PROGRAM S09_CardCarrying
VAR
	//工站
	station					: REFERENCE TO FB_Station:=fbstation[9];
	//气缸
	fbHOZCyl	:REFERENCE TO FB_Cylinder:=fbCylinder[33];	//	卡片上料Y轴气缸
	fbVTCCyl_1	:REFERENCE TO FB_Cylinder:=fbCylinder[34];	//	卡片上料Z轴气缸1(上)
	fbVTCCyl_2	:REFERENCE TO FB_Cylinder:=fbCylinder[35];	//	卡片上料Z轴气缸2（下）



	//伺服
	fbROTAxisMove	 :REFERENCE TO FB_Axis:=fbAxis[16];	//	出料线体伺服
	fbZAxisStepMotor1	 :REFERENCE TO FB_Axis:=fbAxis[17];	//	卡片顶升步进
	fbZAxisStepMotor2	 :REFERENCE TO FB_Axis:=fbAxis[18];	//	卡片顶升步进
	


	
	//延时
	arTonDelay :ARRAY[1..20] OF TON;
	//返回值
	UdiReturnValue :ARRAY[1..20] OF UDINT;
	//过程记录
	tsModuleProcess:ARRAY[1..gc_ModuleProNo] OF DUT_Process;
	xClearModuleProcessDone:BOOL;
	bClearProcessStep	:BYTE;
	i: INT;
	
	// //破真空
	xVacuum_BreakValveControl:ARRAY[1..2]OF BOOL;
	// //破真空完成
	xVacuum_BreakCompleted:ARRAY[1..2] OF BOOL;
	// //卡片到位传感器
	xCardSensorReached: ARRAY[1..2] of bool;
	// //卡片存在检测
	xCardCheckSensor: ARRAY[1..2] of bool;
	
	 //报警屏蔽
	_AlarmDisable: BOOL;
	// //真空吸动作
	xVacuum_WorkValveControl: ARRAY[1..2] OF BOOL;
	// //真空吸到达真空
	xVacuumWorkCompleted:ARRAY[1..2] OF BOOL;
	// //皮带线上检测卡片
	xBeltCardCheckSensor:ARRAY[1..2] OF BOOL;
	// //允许机械手放置深孔板
	xPutBoxPermit: BOOL;
	//首次循环
	_FirstCycle: ARRAY[1..10]OF BOOL;
END_VAR

A_Input();
Alarm();
Delay();
FlowAuto();
FlowInit();
General();
ILC();
TipAuto();
TipManual();
Z_Output();

ACTION A_Input:
//气缸
fbHOZCyl.xWP_Sensor	:=	IxS08HOZCylWP	;
fbHOZCyl.xHP_Sensor	:=	IxS08HOZCylHP	;
fbVTCCyl_1.xWP_Sensor	:=	IxS08VTCCyl_1WP	;
fbVTCCyl_1.xHP_Sensor	:=	IxS08VTCCyl_1HP	;
fbVTCCyl_2.xWP_Sensor	:=	IxS08VTCCyl_2WP	;
fbVTCCyl_2.xHP_Sensor	:=	IxS08VTCCyl_2HP	;
//传感器
xBeltCardCheckSensor[1]:=IxBeltEntryCardCheckSensor1;
xBeltCardCheckSensor[2]:=IxBeltEntryCardCheckSensor2;
END_ACTION

ACTION Alarm:
//
station.adwAlarm[1].00:=station.xInitTimeout;	  			//S09CardCarrying 初始化超时
(*station.adwAlarm[1].01:=TRUE;	  							//S09CardCarrying 卡片不足，需要补充*)
END_ACTION

ACTION Delay:
(*arTonDelay[01](IN:= , PT:=T#0.1S , Q=> , ET=> );*)//TipAuto使用
arTonDelay[02](IN:=  , PT:=T#1S , Q=> , ET=> );
arTonDelay[03](IN:=   , PT:=T#1S , Q=> , ET=> );
arTonDelay[04](IN:= , PT:=T#0.1S , Q=> , ET=> );
arTonDelay[05](IN:= , PT:=T#0.1S , Q=> , ET=> );
arTonDelay[06](IN:= , PT:=T#0.1S , Q=> , ET=> );
arTonDelay[07](IN:= , PT:=T#0.1S , Q=> , ET=> );
arTonDelay[08](IN:= , PT:=T#0.1S , Q=> , ET=> );
arTonDelay[09](IN:= , PT:=T#0.1S , Q=> , ET=> );
END_ACTION

ACTION FlowAuto:

//-----------------------------------------初始化是否完成判断----------------------------------------------
IF NOT station.xInitDone 
THEN
 	station.iStepAuto:=0;
 	station.xDone:=FALSE;
	station.xRunningOffProhibit := FALSE ;//运行中信号Off禁止
ELSIF station.xRunning  
THEN
//-----------------------------------------动作步骤--------------------------------------------------------
CASE station.iStepAuto OF	  
	0: //----Home Step，等待启动----
		IF station.xDisabled 
			AND station.xCanRun 
			AND NOT fbMachine[1].xStopped 
			AND NOT station.xSingleRunning 
		THEN
			station.xDone:=TRUE;
		END_IF
		
		IF  station.xSingleRunning 
			OR station.xCanRun 
			//AND NOT station.xDone 
			AND NOT station.xDisabled 
			AND NOT fbMachine[1].xStopped
		THEN
			station.xCycleEnable:=TRUE;
			//station.xDone:= FALSE;  
			station.iStepAuto:= 10;
		END_IF
    10: //复位数据 
			fbZAxisStepMotor1.xJogForwardAuto:=FALSE;
			fbZAxisStepMotor2.xJogForwardAuto:=FALSE;
			IF  station.xSingleRunning THEN
				 FOR i:=1 TO gc_ModuleProNo BY 1 DO
						 MEMSET(ADR(tsModuleProcess[i]),0,SIZEOF(tsModuleProcess[i]));
				 END_FOR
			END_IF
			station.iStepAuto:=20;
	20://检查卡片是否在位
			_AlarmDisable:=FALSE;
			IF  xCardCheckSensor[1] AND
				xCardCheckSensor[2] THEN
				station.iStepAuto:=30;
 			ELSE
				station.iStepAuto:=25;
			END_IF
	25://卡片缺少,伺服回参考点
			 fbZAxisStepMotor1.xMoveAuto[1]:=TRUE;
			 fbZAxisStepMotor2.xMoveAuto[1]:=TRUE;
			IF    fbZAxisStepMotor1.xMoveInPos[1] AND 
				fbZAxisStepMotor2.xMoveInPos[1] THEN
				station.iStepAuto:=26;
			END_IF
	26://卡片确实报警
			IF NOT  _AlarmDisable  THEN
				station.adwAlarm[1].01:=TRUE;//S09CardCarrying 卡片不足，需要补充
				_AlarmDisable:=TRUE;
			END_IF
				station.iStepAuto:=20;
			
	30://步进上升等待到达传感器
		IF 	NOT 	xCardSensorReached[1]  THEN
			fbZAxisStepMotor1.xJogForwardAuto:=TRUE;
		ELSE
			fbZAxisStepMotor1.xJogForwardAuto:=FALSE;
		END_IF
		IF 	NOT 	xCardSensorReached[2]  THEN
			fbZAxisStepMotor2.xJogForwardAuto:=TRUE;
		ELSE
			fbZAxisStepMotor2.xJogForwardAuto:=FALSE;
		END_IF
		IF  xCardSensorReached[1] AND 
			xCardSensorReached[2] THEN
			station.iStepAuto:=35;
		END_IF
	35://判断流程
		IF  tsModuleProcess[1].xProcessCompleted AND 
			tsModuleProcess[2].xProcessCompleted THEN
			station.iStepAuto:=170;
		ELSE
			station.iStepAuto:=40;
		END_IF
	
		station.iStepAuto:=40;
	40://X轴气缸伸出
		fbHOZCyl.xAuto :=TRUE;
		IF fbHOZCyl.xWP_Delay THEN
			station.iStepAuto:=50;
		END_IF
	50://上Z轴下降
		fbVTCCyl_1.xAuto:=TRUE;
		IF fbVTCCyl_1.xWP_Delay THEN
			station.iStepAuto:=60;	
		END_IF
	60://下Z轴下降
		fbVTCCyl_2.xAuto:=TRUE;
		IF fbVTCCyl_2.xWP_Delay THEN
			station.iStepAuto:=70;	
		END_IF

	70:////Restore_after_Estop_Process1 取卡片流程
			IF tsModuleProcess[1].xProcessNotStarted AND NOT  tsModuleProcess[1].xProcessStarted THEN
					station.iStepAuto :=80; (*process not started*)
			ELSIF  tsModuleProcess[1].xProcessStarted AND NOT  tsModuleProcess[1].xProcessCompleted THEN
				 station.iStepAuto := 80;(*process started*)
			ELSIF  tsModuleProcess[1].xProcessCompleted AND NOT tsModuleProcess[1].xQDataCompleted  THEN
					station.iStepAuto := 105 ;(*process completed*)
			ELSIF tsModuleProcess[1].xQDataCompleted THEN
					station.iStepAuto :=105;(*Qdata completed *)
			ELSE
					station.iStepAuto :=80; 
			END_IF	
	80://
				tsModuleProcess[1].xProcessNotStarted:=TRUE;
				station.iStepAuto:= 90;
	90://真空吸动作
				tsModuleProcess[1].xProcessStarted:=TRUE;
				xVacuum_BreakValveControl[1]:=FALSE;
				xVacuum_BreakValveControl[2]:=FALSE;
				xVacuum_WorkValveControl[1]:=TRUE;
				xVacuum_WorkValveControl[2]:=TRUE;
			IF    xVacuumWorkCompleted[1] AND xVacuumWorkCompleted[2] THEN
				station.iStepAuto:= 100;
			END_IF
	100://真空吸动作完成
			tsModuleProcess[1].xProcessCompleted:=TRUE;
			station.iStepAuto:= 110;
	105://上Z轴上升
			fbVTCCyl_1.xAuto:=FALSE;
		IF fbVTCCyl_1.xHP_Delay THEN
			station.iStepAuto:=110;	
		END_IF
	110:////Restore_after_Estop_Process2 抖动流程
			IF tsModuleProcess[2].xProcessNotStarted AND NOT  tsModuleProcess[2].xProcessStarted THEN
					station.iStepAuto :=130; (*process not started*)
			ELSIF  tsModuleProcess[2].xProcessStarted AND NOT  tsModuleProcess[2].xProcessCompleted THEN
				 station.iStepAuto := 130;(*process started*)
			ELSIF  tsModuleProcess[2].xProcessCompleted AND NOT tsModuleProcess[2].xQDataCompleted  THEN
					station.iStepAuto := 160 ;(*process completed*)
			ELSIF tsModuleProcess[2].xQDataCompleted THEN
					station.iStepAuto :=160;(*Qdata completed *)
			ELSE
					station.iStepAuto :=120; 
			END_IF	
	120://
				tsModuleProcess[2].xProcessNotStarted:=TRUE;
				station.iStepAuto:= 130;
				
	130://	开始抖动流程
				tsModuleProcess[2].xProcessStarted:=TRUE;	
				fbVTCCyl_2.xAuto:=FALSE;
				IF fbVTCCyl_2.xHP_Delay THEN
					station.iStepAuto:=140;	
				END_IF	
	140:		
				fbVTCCyl_2.xAuto:=TRUE;
				IF fbVTCCyl_2.xWP_Delay THEN
					station.iStepAuto:=150;	
				END_IF		
	150://抖动完成
			tsModuleProcess[2].xProcessCompleted:=TRUE;		
			station.iStepAuto:=160;		
	160://下Z轴上升
				fbVTCCyl_2.xAuto:=FALSE;
				IF fbVTCCyl_2.xHP_Delay THEN
					station.iStepAuto:=165;	
				END_IF	
				
	165://检查是否允许放卡片
			IF  NOT xBeltCardCheckSensor[1] AND 
				NOT xBeltCardCheckSensor[2] AND 
				NOT  station.xdone 			AND
				(NOT _FirstCycle[1] OR S10_BeltCarrying.station.xDone )THEN 
				station.iStepAuto:=170;
				_FirstCycle[1]:=TRUE;
			END_IF
	170:////Restore_after_Estop_Process3 放料流程
			IF tsModuleProcess[3].xProcessNotStarted AND NOT  tsModuleProcess[3].xProcessStarted THEN
					station.iStepAuto :=190; (*process not started*)
			ELSIF  tsModuleProcess[3].xProcessStarted AND NOT  tsModuleProcess[3].xProcessCompleted THEN
				 station.iStepAuto := 190;(*process started*)
			ELSIF  tsModuleProcess[3].xProcessCompleted AND NOT tsModuleProcess[3].xQDataCompleted  THEN
					station.iStepAuto := 250 ;(*process completed*)
			ELSIF tsModuleProcess[3].xQDataCompleted THEN
					station.iStepAuto :=250;(*Qdata completed *)
			ELSE
					station.iStepAuto :=180; 
			END_IF	
	180:
				tsModuleProcess[3].xProcessNotStarted:=TRUE;
				station.iStepAuto:= 190;
	190://Y轴回原点
				fbHOZCyl.xAuto:=FALSE;
				IF fbHOZCyl.xHP_Delay THEN
					station.iStepAuto:=200;	
				END_IF		
	200://上Z轴气缸下降
				fbVTCCyl_1.xAuto:=TRUE;
				IF fbVTCCyl_1.xWP_Delay THEN
					station.iStepAuto:=210;	
				END_IF							
	220://下Z轴气缸下降
				fbVTCCyl_2.xAuto:=TRUE;
				IF fbVTCCyl_2.xWP_Delay THEN
					station.iStepAuto:=230;	
				END_IF			
	230://破真空
				tsModuleProcess[3].xProcessStarted:=TRUE;
			   xVacuum_BreakValveControl[1]:=TRUE;
				xVacuum_BreakValveControl[2]:=TRUE;
				xVacuum_WorkValveControl[1]:=FALSE;
				xVacuum_WorkValveControl[2]:=FALSE;
			IF   xVacuum_BreakCompleted[1] AND 
				 xVacuum_BreakCompleted[2] THEN
				 xVacuum_BreakValveControl[1]:=FALSE;
				 xVacuum_BreakValveControl[2]:=FALSE;
				 station.iStepAuto:=240;		
			END_IF
	240://流程完成
				tsModuleProcess[3].xProcessCompleted:=TRUE;
				 station.iStepAuto:=250;
	250://上Z轴上升
				fbVTCCyl_1.xAuto:=FALSE;
				IF fbVTCCyl_1.xHP_Delay THEN
					station.iStepAuto:=260;	
				END_IF
	260://下Z轴上升
				fbVTCCyl_2.xAuto:=FALSE;
				IF fbVTCCyl_2.xHP_Delay THEN
					station.iStepAuto:=270;	
				END_IF
	270://检查卡片检测是否在位
		IF  xBeltCardCheckSensor[1] AND 
			xBeltCardCheckSensor[2] THEN
			 station.iStepAuto:=280;
		END_IF
	280://允许放置深孔板
			station.iStepAuto:=290;
	290://清除过程数据
			FOR i:=1 TO gc_ModuleProNo BY 1 DO
				MEMSET(ADR(tsModuleProcess[i]),0,SIZEOF(tsModuleProcess[i]));
			END_FOR
			station.iStepAuto:=999;
			
	999://----Single Run Finish----
			
		station.iStepAuto :=0;
		IF NOT station.xSingleContinuousRun THEN
			station.xSingleRunFlag:=FALSE;
		END_IF
		
		station.xCycleEnable:=FALSE;	
		station.xDone:=TRUE;
	ELSE
		;	
END_CASE
(*******************************步进上载卡片*****************************)


END_IF
END_ACTION

ACTION FlowInit:
IF NOT station.xIniting THEN
  station.iStepInit:=0;    
ELSE
//--------------------------------------------初始化步序----------------------------------
CASE station.iStepInit OF	
 0://  
  	IF station.xIniting THEN	
  	  station.iStepInit:=10;	
  	END_IF	
10://复位数据
	station.iStepInit:=999;
//20://检查是否需要破真空	
//	IF tsModuleProcess[1].xProcessStarted AND
//		 NOT tsModuleProcess[1].xProcessCompleted THEN
//		 station.iStepInit:=30;
//	ELSE
//		station.iStepInit:=40;	
//	END_IF
//30://破真空
//		xVacuum_WorkValveControl[1]:=FALSE;
//		xVacuum_WorkValveControl[2]:=FALSE;
//		xVacuum_BreakValveControl[1]:=TRUE;
//		xVacuum_BreakValveControl[2]:=TRUE;
//	IF   xVacuum_BreakCompleted[1] AND 
//		 xVacuum_BreakCompleted[2] THEN
//		 xVacuum_BreakValveControl[1]:=FALSE;
//		 xVacuum_BreakValveControl[2]:=FALSE;
//		 station.iStepInit:=40;	
//	END_IF
//40://上Z轴上升
//	fbVTCCyl_1.xInit:=TRUE;
//	IF  fbVTCCyl_1.xHP_Delay THEN
//		station.iStepInit:=50;	
//	END_IF
//50://下轴上升
//	fbVTCCyl_2.xInit:=TRUE;
//	IF  fbVTCCyl_2.xHP_Delay THEN
//		station.iStepInit:=60;	
//	END_IF
//60://X轴气缸回原
//	fbHOZCyl.xInit:=TRUE;
//	IF  fbHOZCyl.xHP_Delay THEN
//		station.iStepInit:=70;	
//	END_IF		
//70://卡片步进上电
//	fbZAxisStepMotor1.xPowerInit:=TRUE;
//	fbZAxisStepMotor2.xPowerInit:=TRUE;
//	IF		fbZAxisStepMotor1.xPowerOn AND
//		    fbZAxisStepMotor2.xPowerOn THEN
//			station.iStepInit:=80;	
//	END_IF
//80://回原点
//	fbZAxisStepMotor1.xReferenceAuto:=TRUE;
//	fbZAxisStepMotor2.xReferenceAuto:=TRUE;
//	station.iStepinit:=90;
//90:
//   IF  fbAxisHome[17].home_done  AND 
//		fbAxisHome[18].home_done THEN 
//		 fbZAxisStepMotor1.xReferenceAuto:=FALSE;
//		fbZAxisStepMotor2.xReferenceAuto:=FALSE;
//		 station.iStepInit:=100;  
//	END_IF
//100://去待机位置
//	 fbZAxisStepMotor1.xMoveAuto[1]:=TRUE;
//	  fbZAxisStepMotor2.xMoveAuto[1]:=TRUE;
//	IF    fbZAxisStepMotor1.xMoveInPos[1] AND 
//		fbZAxisStepMotor2.xMoveInPos[1] THEN
//		 station.iStepInit:=999;  
//	END_IF
999://初始化完成	
	station.iStepInit:=0;
	station.xInitDone:=TRUE;  
END_CASE
END_IF
END_ACTION

ACTION General:

END_ACTION

ACTION ILC:

//---------------------------------------------------工站可执行-------------------------------------------------------
station.xCanRun :=TRUE ;

//---------------------------------------------------气缸动作条件-------------------------------------------

fbHOZCyl.xOffILC	:=	TRUE;//fbVTCCyl_1.xHP_Delay AND  fbVTCCyl_1.xHP_Delay 	;
fbHOZCyl.xOnILC		:=	TRUE;//fbVTCCyl_1.xHP_Delay AND  fbVTCCyl_1.xHP_Delay	;
fbVTCCyl_1.xOffILC	:=	TRUE;//fbHOZCyl.xHP_Delay OR fbHOZCyl.xWP_Delay	;
fbVTCCyl_1.xOnILC	:=	TRUE;//fbHOZCyl.xHP_Delay OR fbHOZCyl.xWP_Delay	;
fbVTCCyl_2.xOffILC	:=	TRUE	;
fbVTCCyl_2.xOnILC	:=	TRUE; //fbHOZCyl.xHP_Delay OR fbHOZCyl.xWP_Delay	;


//---------------------------------------------------伺服动作条件-------------------------------------------


fbZAxisStepMotor1.xRunILC := 
fbZAxisStepMotor1.xMoveILC[1] :=
fbZAxisStepMotor1.xMoveILC[2] :=
fbZAxisStepMotor1.xMoveILC[3] :=
fbZAxisStepMotor1.xMoveILC[4] :=
fbZAxisStepMotor1.xMoveILC[5] := TRUE ;


fbZAxisStepMotor2.xRunILC := 
fbZAxisStepMotor2.xMoveILC[1] :=
fbZAxisStepMotor2.xMoveILC[2] :=
fbZAxisStepMotor2.xMoveILC[3] :=
fbZAxisStepMotor2.xMoveILC[4] :=
fbZAxisStepMotor2.xMoveILC[5] := TRUE ;
END_ACTION

ACTION TipAuto:

//------------------------------------------------AutoTip Cylinder--------------------------------
station.adwAutoTip[1].00	:=	fbHOZCyl.xAutoTip	;
station.adwAutoTip[1].01	:=	fbVTCCyl_1.xAutoTip	;
station.adwAutoTip[1].02	:=	fbVTCCyl_2.xAutoTip	;	
//------------------------------------------------AutoTip Servo--------------------------------
//**************************************
FOR i:= 1 TO 5 BY 1 DO 
	IF fbROTAxisMove.xMoveAuto[i] THEN
		fbROTAxisMove.iPosNumber := i ;
	END_IF
	IF fbZAxisStepMotor1.xMoveAuto[i] THEN
		fbZAxisStepMotor1.iPosNumber := i ;
	END_IF
	IF fbZAxisStepMotor2.xMoveAuto[i] THEN
		fbZAxisStepMotor2.iPosNumber := i ;
	END_IF
	
END_FOR


IF  fbMachine[1].xAutoMode AND NOT fbMachine[1].xRunning  THEN
	  arTonDelay[01](IN:=True , PT:=T#1S , Q=> , ET=> );
else
	  arTonDelay[01](IN:=false);
END_IF
IF arTonDelay[1].Q  THEN 
IF	fbROTAxisMove.iPosNumber=1 	AND NOT fbROTAxisMove.xMoveInPos[1] 	THEN 	station.adwAutoTip[1].10:=TRUE	;	END_IF//轴伺服自动时位置不在位置1
if	fbROTAxisMove.iPosNumber=2	AND NOT fbROTAxisMove.xMoveInPos[2]	THEN 	station.adwAutoTip[1].11:=TRUE	;	END_IF//轴伺服自动时位置不在位置2
if	fbROTAxisMove.iPosNumber=3	AND NOT fbROTAxisMove.xMoveInPos[3]	THEN 	station.adwAutoTip[1].12:=TRUE	;	END_IF//轴伺服自动时位置不在位置3
if	fbROTAxisMove.iPosNumber=4	AND NOT fbROTAxisMove.xMoveInPos[4]	THEN 	station.adwAutoTip[1].13:=TRUE	;	END_IF//轴伺服自动时位置不在位置4
if	fbROTAxisMove.iPosNumber=5	AND NOT fbROTAxisMove.xMoveInPos[5]	THEN 	station.adwAutoTip[1].14:=TRUE	;	END_IF//轴伺服自动时位置不在位置5
if	fbZAxisStepMotor1.iPosNumber=1 	AND NOT fbZAxisStepMotor1.xMoveInPos[1] 	THEN 	station.adwAutoTip[1].15:=TRUE	;	END_IF//轴伺服自动时位置不在位置1
if	fbZAxisStepMotor1.iPosNumber=2	AND NOT fbZAxisStepMotor1.xMoveInPos[2]	THEN 	station.adwAutoTip[1].16:=TRUE	;	END_IF//轴伺服自动时位置不在位置2
if	fbZAxisStepMotor1.iPosNumber=3	AND NOT fbZAxisStepMotor1.xMoveInPos[3]	THEN 	station.adwAutoTip[1].17:=TRUE	;	END_IF//轴伺服自动时位置不在位置3
if	fbZAxisStepMotor1.iPosNumber=4	AND NOT fbZAxisStepMotor1.xMoveInPos[4]	THEN 	station.adwAutoTip[1].18:=TRUE	;	END_IF//轴伺服自动时位置不在位置4
if	fbZAxisStepMotor1.iPosNumber=5	AND NOT fbZAxisStepMotor1.xMoveInPos[5]	THEN 	station.adwAutoTip[1].19:=TRUE	;	END_IF//轴伺服自动时位置不在位置5
if	fbZAxisStepMotor2.iPosNumber=1 	AND NOT fbZAxisStepMotor2.xMoveInPos[1] 	THEN 	station.adwAutoTip[1].20:=TRUE	;	END_IF//轴伺服自动时位置不在位置1
if	fbZAxisStepMotor2.iPosNumber=2	AND NOT fbZAxisStepMotor2.xMoveInPos[2]	THEN 	station.adwAutoTip[1].21:=TRUE	;	END_IF//轴伺服自动时位置不在位置2
if	fbZAxisStepMotor2.iPosNumber=3	AND NOT fbZAxisStepMotor2.xMoveInPos[3]	THEN 	station.adwAutoTip[1].22:=TRUE	;	END_IF//轴伺服自动时位置不在位置3
if	fbZAxisStepMotor2.iPosNumber=4	AND NOT fbZAxisStepMotor2.xMoveInPos[4]	THEN 	station.adwAutoTip[1].23:=TRUE	;	END_IF//轴伺服自动时位置不在位置4
if	fbZAxisStepMotor2.iPosNumber=5	AND NOT fbZAxisStepMotor2.xMoveInPos[5]	THEN 	station.adwAutoTip[1].24:=TRUE	;	END_IF//轴伺服自动时位置不在位置5

	
		
END_IF
END_ACTION

ACTION TipManual:
//--------------------------------------------ManualTip------------------------------------------------------

//-------------------------------------------气缸提示---------------------------------------------------------




/////////////////////////////////////////////////////////////////////////////////////////////////////////////////
END_ACTION

ACTION Z_Output:
(**************************气缸输出********************************)
QxS08HOZCylWP	:=	fbHOZCyl.xWP_Valve	;
QxS08HOZCylHP	:=	fbHOZCyl.xHP_Valve	;
QxS08VTCCyl_1WP	:=	fbVTCCyl_1.xWP_Valve	;
QxS08VTCCyl_1HP	:=	fbVTCCyl_1.xHP_Valve	;
QxS08VTCCyl_2WP	:=	fbVTCCyl_2.xWP_Valve	;
QxS08VTCCyl_2HP	:=	fbVTCCyl_2.xHP_Valve	;
END_ACTION

END_PROGRAM

(* stored: Version 1.1.0.1, ProductVersion 3.1.4024.9
   POU S09_CardCarrying: Id {719670c2-0d20-4660-9913-c0a0e65d6f7c}, SpecialFunc None
   Action A_Input: Id {ba23078b-8967-4278-88bc-5ab193e99c06}
   Action Alarm: Id {0a31e6b9-e40b-403d-b500-5fe16c4985f5}
   Action Delay: Id {7954a2d3-613f-47d1-88d7-daa2a45cb229}
   Action FlowAuto: Id {cc7578fa-0edf-4606-8ba0-a269ab7b1135}
   Action FlowInit: Id {0430a122-4c62-44ac-9816-5c9a71171d9e}
   Action General: Id {45030b2b-c41a-4da3-bcf2-db15989ba868}
   Action ILC: Id {c76333f4-12c7-4311-b266-a45dd1caf128}
   Action TipAuto: Id {95719469-7bab-4353-9341-e6e5d4586814}
   Action TipManual: Id {bfbca7f7-f29c-4c3f-9863-da81fea994f1}
   Action Z_Output: Id {e5141706-d276-488d-8e03-6fb5bac7b25e} *)
